/// This enumeration contains all steps that are used by the various sequences of a unit.
/// Sequences use a subrange (***Begin to ***End) of this enumeration.
{attribute 'qualified_only'}
{attribute 'to_string'}
TYPE ScriblyStep :
(
  Undefined := 0
  
  ,BootBegin
  ,BootEnd 

  ,StopBegin
  ,StopEnd

  ,AutomaticBegin
  ,AutomaticWaitSegment
  ,AutomaticMoveToSegmentStart
  ,AutomaticMovePenDown
  ,AutomaticDraw
  ,AutomaticMovePenUp
  ,AutomaticDrawLine
  ,AutomaticDrawCatmulRomDrawSplineBegin
  ,AutomaticDrawCatmulRomDrawSpline
  ,AutomaticEnd
  
  ,GoHomeBegin
  ,GoHomeMoveUp  
  ,GoHomeReferenceXY
  ,GoHomeEnd 
  
  ,FaultReactionBegin
  ,FaultReactionEnd
);
END_TYPE

(* stored: Version 1.1.0.1
   DUT ScriblyStep: Id {3b1cca9d-d18b-4c44-8357-8b848a0bc3fb} *)
